// TIA Portal V16 export
// export: Created 2023-03-29T11:03:28.8305477Z, ExportSetting WithDefaults, DisplayName Totally Integrated Automation Portal, DisplayVersion V16 Update 6, DisplayName TIA Portal Version Control Interface, DisplayVersion V16 Update 2, DisplayName TIA Portal Openness, DisplayVersion V16 Update 6, DisplayName STEP 7 Professional, DisplayVersion V16 Update 6, DisplayName STEP 7 Safety, DisplayVersion V16, DisplayName WinCC Advanced, DisplayVersion V16 Update 6
FUNCTION "Detection_Changes_Data_Real" : Void   // FC33, LAD
{ S7_Optimized_Access := 'TRUE' }
AUTHOR : rtecmer
VERSION : 0.1
// Funkcja porównuje wartości w bloku wymiany danych i jeśli zaszła zmiana wprowadza ją
// stored: AutoNumber true, IsIECCheckEnabled false, SetENOAutomatically false, UDAEnableTagReadback false
   VAR_IN_OUT
      "tempdbHold_SendingTCP.sterowanie." : Real;   // zadana wartośc zmiennej do porównania
      "DB10_instance_SCADA." : Real;   // zmienna w db której porównujemy
      memRisingTriger_Data_ : Bool;   // bit pamięci zbocza zmiany
      "dbHold_Sending.data.stat.control." : Real;   // zmienna w db wyjścia do zmiany
   END_VAR
   VAR_TEMP   // added for the SCL form of the ladder/FBD networks
      _w1 : Bool;
      _w2 : Bool;
   END_VAR
BEGIN

REGION Network 1: bit inicjacji wysłąnia nowej wartości
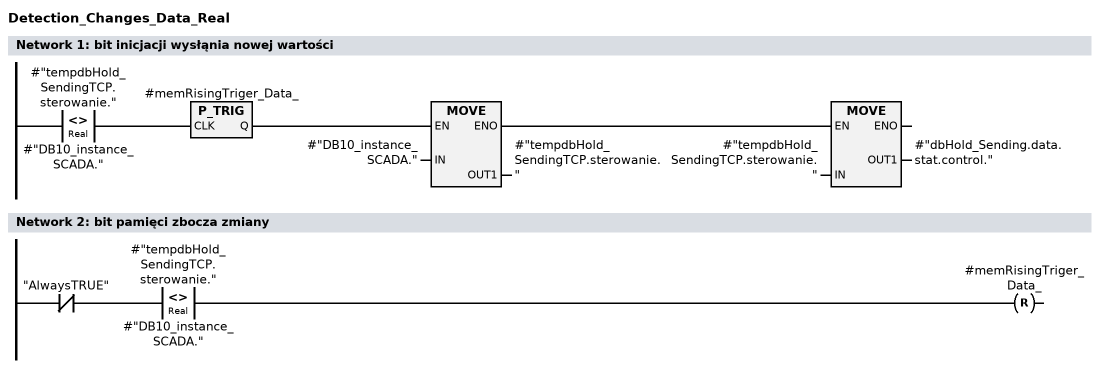
   RUNG wire#powerrail
      { S7_Templates := "SrcType := Real" } NE_Contact(in1 := #"tempdbHold_SendingTCP.sterowanie.", in2 := #"DB10_instance_SCADA.")
      P_Trig( #memRisingTriger_Data_ )
      Move(in := #"DB10_instance_SCADA.", out1 => #"tempdbHold_SendingTCP.sterowanie.")
      Move(in := #"tempdbHold_SendingTCP.sterowanie.", out1 => #"dbHold_Sending.data.stat.control.")
   END_RUNG
   // the same network as SCL:
   #_w1 := #"tempdbHold_SendingTCP.sterowanie." <> #"DB10_instance_SCADA.";
   #_w2 := #_w1 AND NOT #memRisingTriger_Data_;   // rising edge
   #memRisingTriger_Data_ := #_w1;
   IF #_w2 THEN
       #"tempdbHold_SendingTCP.sterowanie." := #"DB10_instance_SCADA.";
       #"dbHold_Sending.data.stat.control." := #"tempdbHold_SendingTCP.sterowanie.";
   END_IF;
END_REGION

REGION Network 2: bit pamięci zbocza zmiany
   RUNG wire#powerrail
      I_Contact( "AlwaysTRUE" )
      { S7_Templates := "SrcType := Real" } NE_Contact(in1 := #"tempdbHold_SendingTCP.sterowanie.", in2 := #"DB10_instance_SCADA.")
      R_Coil( #memRisingTriger_Data_ )
   END_RUNG
   // the same network as SCL:
   IF NOT "AlwaysTRUE" AND (#"tempdbHold_SendingTCP.sterowanie." <> #"DB10_instance_SCADA.") THEN
       #memRisingTriger_Data_ := FALSE;
   END_IF;
END_REGION
END_FUNCTION
